FUNCTION_BLOCK AOI_AxisAdmin
VAR_INPUT
    Enable: BOOL;
	JogN: BOOL;
	JogP: BOOL;
	MoveAbsolute: BOOL;
	MoveRealtive: BOOL;
END_VAR
VAR_OUTPUT
END_VAR
VAR
	MC_Power_Axis: MC_Power;
	MC_Home_Axis: MC_Home;
	MC_MoveAbsolute_Axis: MC_MoveAbsolute;
	MC_MoveAdditive_Axis: MC_MoveAdditive;
	MC_Jog_Axis: MC_Jog;
	MC_Reset_Axis: MC_Reset;
	MC_MoveVelocity_Axis: MC_MoveVelocity;
	MC_Stop_Axis: MC_Stop;
	MC_ReadActualPosition_Axis: MC_ReadActualPosition;
	MC_SetPosition_Axis: MC_SetPosition;
	MC_MoveHome: MC_MoveAbsolute;
	R_TRIG_Home: R_TRIG;
	F_TRIG_Home: F_TRIG;
	MC_CamOut_Axis: MC_CamOut;;
	MC_Power_Stop: MC_Stop;
	MC_GearOut_Axis: mc_gearout;
	MC_MoveRelative_Axis: MC_MoveRelative;
	
	i: INT;
END_VAR
VAR_IN_OUT
	Admin: UDT_AxisAdmin;
END_VAR

IF admin.i.Disable THEN
   Disable();   
END_IF
IF admin.i.mode=0 THEN
   Enable:=FALSE;
   JogN:=FALSE;
   JogP:=FALSE;
   MoveAbsolute:=FALSE;
   MoveRealtive:=FALSE;
END_IF

Homing();
Jog();
MoveAbs();
MoveAdd();
MoveReal();
PowerOn();
Reset();
SetPos();
Stop();
Cam();
admin.o.Active:=MC_MoveAbsolute_Axis.Active OR MC_MoveAdditive_Axis.Active;
IF NOT admin.i.MoveAbs  AND NOT admin.i.MoveAdd AND NOT admin.i.MoveReal THEN
	admin.o.CmdDone:=FALSE;
END_IF
admin.Axis.ReadStatus();
admin.o.Homed:=admin.Axis.Status.Homed;
admin.o.ActPos:=admin.Axis.NcToPlc.ActPos;
admin.o.ActModuloPos:=admin.Axis.NcToPlc.ModuloActPos;
admin.o.ActVel:=admin.Axis.NcToPlc.ActVelo;
admin.o.ActTorq:=admin.Axis.NcToPlc.ActTorque;
admin.o.ErrorID:=admin.Axis.NcToPlc.ErrorCode;

admin.o.InSync:=admin.axis.Status.Coupled;
admin.o.StandStill:=admin.axis.Status.NotMoving;
admin.o.PowerOn:=admin.axis.NcToPlc.StateDWord.20;

IF admin.Axis.Status.Error  OR MC_MoveAbsolute_Axis.Error OR MC_MoveAdditive_Axis.Error OR MC_Jog_Axis.Error OR MC_MoveVelocity_Axis.Error
OR MC_MoveHome.Error OR MC_CamOut_Axis.Error OR MC_Power_Stop.Error OR MC_GearOut_Axis.Error OR MC_MoveRelative_Axis.Error  THEN
   admin.o.Error:=TRUE;
END_IF
IF admin.i.Reset THEN
   admin.o.Error:=FALSE; 
END_IF

FOR i:=1 TO 8 DO
	IF  admin.i.PosRangeTable[i][1] < admin.Axis.NcToPlc.ModuloActPos AND
        admin.Axis.NcToPlc.ModuloActPos < admin.i.PosRangeTable[i][2] THEN
		admin.o.PosInRange[i]:=TRUE;
		ELSE	
		admin.o.PosInRange[i]:=FALSE;
	END_IF
END_FOR

ACTION Cam:
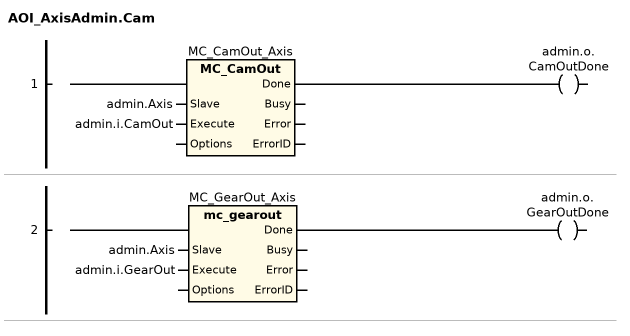
// NETWORK 1
MC_CamOut_Axis(Slave := admin.Axis, Execute := admin.i.CamOut); // MC_CamOut
admin.o.CamOutDone := MC_CamOut_Axis.Done;

// NETWORK 2
MC_GearOut_Axis(Slave := admin.Axis, Execute := admin.i.GearOut); // mc_gearout
admin.o.GearOutDone := MC_GearOut_Axis.Done;
END_ACTION

ACTION Disable:
Admin.i.CamIn:=FALSE;
Admin.i.CamOut:=FALSE;
Admin.i.Enable:=FALSE;
Admin.i.GearIn:=FALSE;
Admin.i.GearOut:=FALSE;
Admin.i.MoveAbs:=FALSE;
Admin.i.MoveAdd:=FALSE;
Admin.i.MoveVel:=FALSE;
Admin.i.JogN:=FALSE;
Admin.i.JogP:=FALSE;
Admin.i.Stop:=FALSE;
Admin.i.Home:=FALSE;
Admin.i.Reset:=FALSE;
Admin.i.SelectCamTable:=FALSE;
Admin.i.SetPosExe:=FALSE;
Admin.i.Disable:=FALSE;
Admin.i.MoveReal:=FALSE;
END_ACTION

ACTION Homing:
IF admin.i.HomeMode=0 OR admin.i.HomeMode=1 THEN
	MC_Home_Axis.HomingMode:=MC_DefaultHoming;
END_IF

IF admin.i.HomeMode=2  THEN
   MC_Home_Axis.HomingMode:=MC_Direct;
END_IF

MC_Home_Axis(
	Axis:=Admin.Axis , 
	Execute:=admin.i.Home AND admin.o.PowerOn , 
	Position:=admin.i.HomeOffset , 
	HomingMode:= , 
	BufferMode:= , 
	Options:= , 
	bCalibrationCam:= admin.i.HomeCali, 
	Done=> admin.o.HomeDone, 
	Busy=> , 
	Active=> , 
	CommandAborted=> , 
	Error=> , 
	ErrorID=> );
END_ACTION

ACTION Jog:
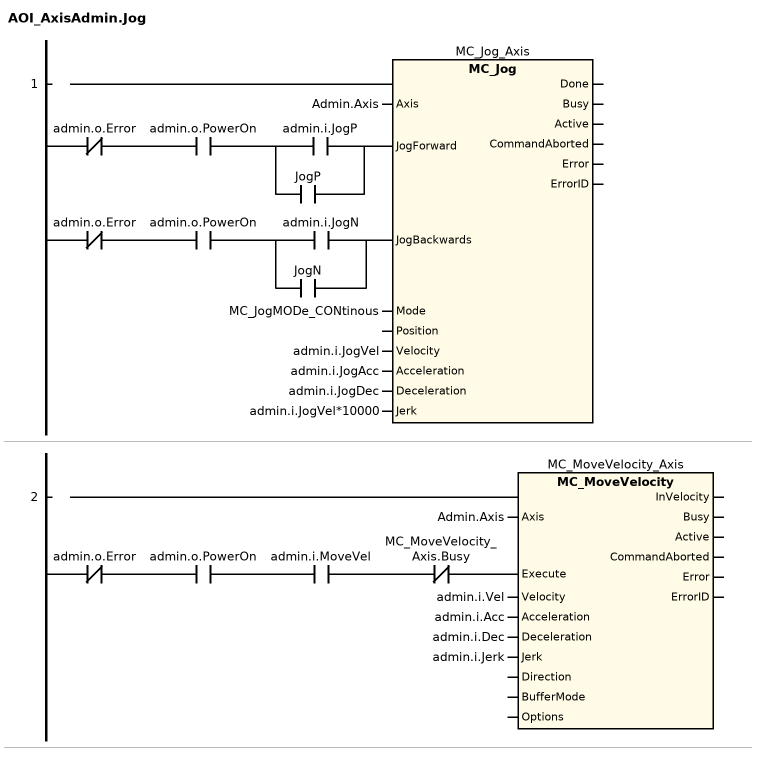
// NETWORK 1
MC_Jog_Axis(
    Axis := Admin.Axis,
    JogForward := NOT admin.o.Error AND admin.o.PowerOn AND (admin.i.JogP OR JogP),
    JogBackwards := NOT admin.o.Error AND admin.o.PowerOn AND (admin.i.JogN OR JogN),
    Mode := MC_JogMODe_CONtinous,
    Velocity := admin.i.JogVel,
    Acceleration := admin.i.JogAcc,
    Deceleration := admin.i.JogDec,
    Jerk := admin.i.JogVel*10000); // MC_Jog

// NETWORK 2
MC_MoveVelocity_Axis(
    Axis := Admin.Axis,
    Execute := NOT admin.o.Error AND admin.o.PowerOn AND admin.i.MoveVel AND NOT MC_MoveVelocity_Axis.Busy,
    Velocity := admin.i.Vel,
    Acceleration := admin.i.Acc,
    Deceleration := admin.i.Dec,
    Jerk := admin.i.Jerk); // MC_MoveVelocity
END_ACTION

ACTION MoveAbs:
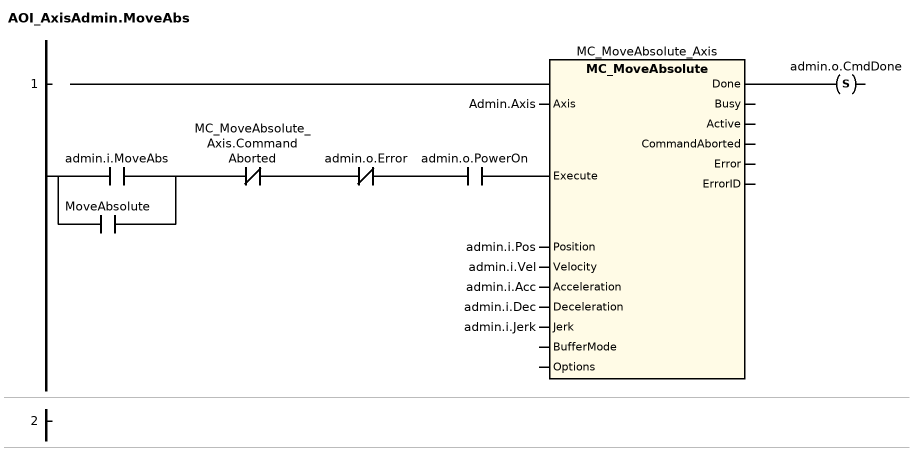
// NETWORK 1
MC_MoveAbsolute_Axis(
    Axis := Admin.Axis,
    Execute := (admin.i.MoveAbs OR MoveAbsolute) AND NOT MC_MoveAbsolute_Axis.CommandAborted AND NOT admin.o.Error AND admin.o.PowerOn,
    Position := admin.i.Pos,
    Velocity := admin.i.Vel,
    Acceleration := admin.i.Acc,
    Deceleration := admin.i.Dec,
    Jerk := admin.i.Jerk); // MC_MoveAbsolute
admin.o.CmdDone S= MC_MoveAbsolute_Axis.Done;

// NETWORK 2
END_ACTION

ACTION MoveAdd:
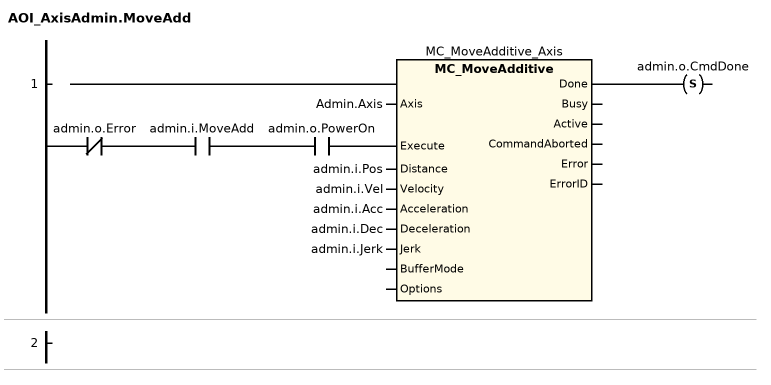
// NETWORK 1
MC_MoveAdditive_Axis(
    Axis := Admin.Axis,
    Execute := NOT admin.o.Error AND admin.i.MoveAdd AND admin.o.PowerOn,
    Distance := admin.i.Pos,
    Velocity := admin.i.Vel,
    Acceleration := admin.i.Acc,
    Deceleration := admin.i.Dec,
    Jerk := admin.i.Jerk); // MC_MoveAdditive
admin.o.CmdDone S= MC_MoveAdditive_Axis.Done;

// NETWORK 2
END_ACTION

ACTION MoveReal:
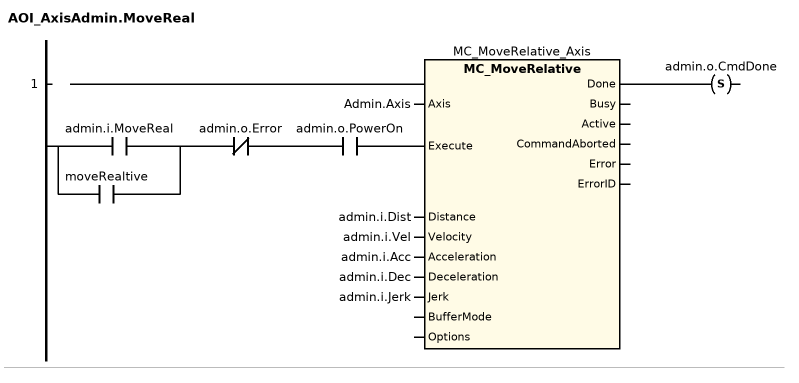
// NETWORK 1
MC_MoveRelative_Axis(
    Axis := Admin.Axis,
    Execute := (admin.i.MoveReal OR moveRealtive) AND NOT admin.o.Error AND admin.o.PowerOn,
    Distance := admin.i.Dist,
    Velocity := admin.i.Vel,
    Acceleration := admin.i.Acc,
    Deceleration := admin.i.Dec,
    Jerk := admin.i.Jerk); // MC_MoveRelative
admin.o.CmdDone S= MC_MoveRelative_Axis.Done;
END_ACTION

ACTION PowerOn:
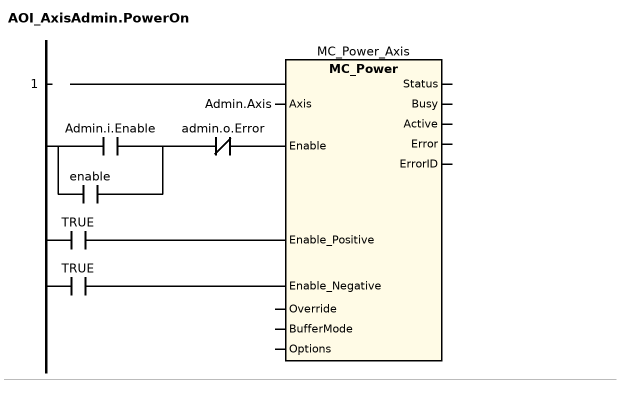
// NETWORK 1
MC_Power_Axis(
    Axis := Admin.Axis,
    Enable := (Admin.i.Enable OR enable) AND NOT admin.o.Error,
    Enable_Positive := TRUE,
    Enable_Negative := TRUE); // MC_Power
END_ACTION

ACTION Reset:
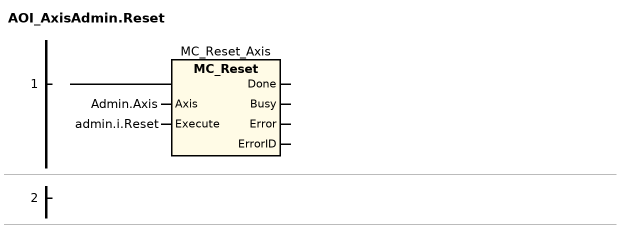
// NETWORK 1
MC_Reset_Axis(Axis := Admin.Axis, Execute := admin.i.Reset); // MC_Reset

// NETWORK 2
END_ACTION

ACTION SetPos:
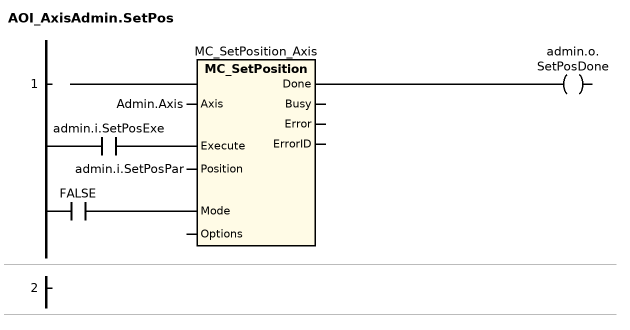
// NETWORK 1
MC_SetPosition_Axis(
    Axis := Admin.Axis,
    Execute := admin.i.SetPosExe,
    Position := admin.i.SetPosPar,
    Mode := FALSE); // MC_SetPosition
admin.o.SetPosDone := MC_SetPosition_Axis.Done;

// NETWORK 2
END_ACTION

ACTION Stop:
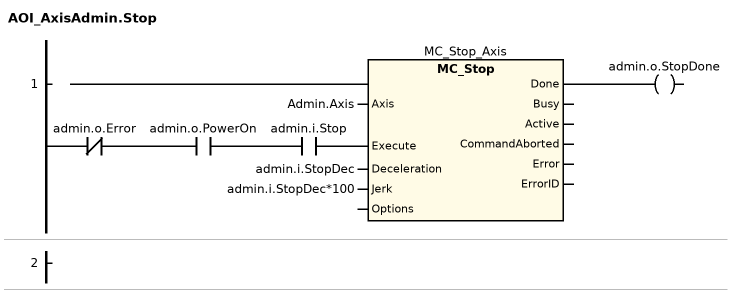
// NETWORK 1
MC_Stop_Axis(
    Axis := Admin.Axis,
    Execute := NOT admin.o.Error AND admin.o.PowerOn AND admin.i.Stop,
    Deceleration := admin.i.StopDec,
    Jerk := admin.i.StopDec*100); // MC_Stop
admin.o.StopDone := MC_Stop_Axis.Done;

// NETWORK 2
END_ACTION

END_FUNCTION_BLOCK

(* stored: Version 1.1.0.1, ProductVersion 3.1.4022.16
   POU AOI_AxisAdmin: Id {92e2bc02-2d46-449e-b721-96a2992fd0b1}, SpecialFunc None
   Action Cam: Id {3d0ecd19-0d22-4c09-8110-17c6e71cb19f}
   Action Disable: Id {24ceca3a-4d58-4318-a9d4-c98bf96c0872}
   Action Homing: Id {a1045205-e522-49ca-8b91-9a4e4d08a148}
   Action Jog: Id {079cd750-2667-4001-9b11-8880874f34b1}
   Action MoveAbs: Id {85e510eb-d73e-4243-91b1-a297d416cbf3}
   Action MoveAdd: Id {97b82c83-74ec-417c-b2c3-68192c881fd0}
   Action MoveReal: Id {3b33f952-8209-46b2-bb6a-9ca700875af0}
   Action PowerOn: Id {d34c23b1-2a07-4fec-ae7a-3391a3d12041}
   Action Reset: Id {666884e7-4067-48b0-bcf1-4587b37433da}
   Action SetPos: Id {14deb118-ca2d-4bde-8e46-58092f317b87}
   Action Stop: Id {39348f77-e705-45e2-90b1-8b2bce02bf76} *)
